TYPE JsonNode :
STRUCT
  Name : STRING;
  Next : POINTER TO JsonNode;
  Child : POINTER TO JsonNode;
  Element : POINTER TO JsonElement;
END_STRUCT
END_TYPE

(* stored: Version 1.1.0.1, ProductVersion 3.1.4024.12
   DUT JsonNode: Id {a7ff27e2-e209-4cf2-9b64-669f247284b6} *)
